PROGRAM prgBattery
VAR PERSISTENT
	bEnableBattery				: BOOL;							//{#lynus.ag#()}
	byPrioBattery				: BYTE;							//{#lynus.ag#()}
	lrMaxCapacityBattery		: LREAL;						//{#lynus.ag#()}
	lrCounterBattProd			: LREAL;						//{#lynus.ag#()}
	lrCounterBattCons			: LREAL;						//{#lynus.ag#()}
	str_IP						: STRING(15):='10.11.90.140';
	m_manual_LoadLimiting: BOOL :=TRUE;
	real_Max_ChargePower: REAL := 30000;
END_VAR
VAR
	fbBattery					: FB_Xelectrix_Powerbox_v2T;
	fbBattCounter				: FB_EnergyCounter;
	bIsEnabledBattery			: BOOL;							//{#lynus.ag#()}
	bResetBattery				: BOOL;							//{#lynus.ag#()}
	bSResetBattery				: BOOL;							//{#lynus.ag#()}
	byErrorWarningBattery		: BYTE;							//{#lynus.ag#()}
	dwSOCBattery				: DWORD;						//{#lynus.ag#()}
	rTargetPowerBattery			: REAL;							//{#lynus.ag#()}
	lrPowerBattery				: LREAL;						//{#lynus.ag#()}
	lrActualCapacityBattery		: LREAL;						//{#lynus.ag#()}
	mtest: BOOL;
	x: REAL;
	byBatteryModbusError: BOOL;									//{#lynus.ag#()}
	lrBatteryCons				: LREAL;							//{#lynus.ag#()}
	lrBatteryProd				: LREAL;							//{#lynus.ag#()}
	FB_Linear_MaxChargePower	: FB_LinearEquation;
	FB_Ramp_Max_Charging_Power	: FB_RAMP;
	FB_Linear_MaxChargePowerSOC	: FB_LinearEquation;
	
END_VAR

IF mtest THEN
	Lynus_Standards.GVL_Energy.stDataOfBatteryInverters[1,1].rTargetPowerEMS:=x;
END_IF

fbBattery(
	bEnable:= bEnableBattery, 
	bActivateControl:=TRUE , 
	byUnitID:= 1, 
	byPriority:= byPrioBattery, 
	diNrOfEMS_IN:= prgEMS.fbEMS.diNrOfEMS_OUT, 
	lrMaxCapacityBattery:= lrMaxCapacityBattery, 
	sIPAdress:= str_IP, 						// modify IP Adress
	bReset:= bResetBattery, 
	m_ManualSetpointEnable:= , 
	i_SetpointPower_Manual_kW:= , 
	m_ManualChargeDischargeMax:= m_manual_LoadLimiting, 
	r_MaxChargePower_W:= real_Max_ChargePower, 
	r_MaxDischargePower_W:= 80000, 
	stDataXelectrix=> , 
	stDataBatt=> , 
	stDataBattInverter=> , 
	stDataEMPower_Grid=> , 
	stDataEMCounter_Grid=> , 
	diNrOfBatt_OUT=> , 
	diNrOfBattInverter_OUT=> , 
	diNrOfEM_OUT_Grid=> , 
	lrMaxCapacityBattery_OUT=> , 
	iSetpointPower_Info=> );

//Out
bIsEnabledBattery := fbBattery.stDataBatt.bEnabled;
bSResetBattery := fbBattery.stDataBattInverter.bStateReset;
dwSOCBattery := fbBattery.stDataBatt.dwSOC;
rTargetPowerBattery := fbBattery.stDataBattInverter.rTargetPower;
lrPowerBattery := fbBattery.stDataBatt.lrPower;
lrActualCapacityBattery := fbBattery.lrMaxCapacityBattery_OUT;	
byErrorWarningBattery := fbBattery.stDataBatt.byErrorWarning;
byBatteryModbusError := fbBattery.stDataXelectrix.eErrorState = 1;
lrBatteryCons := fbBattery.stDataBatt.lrPowerConsumption;
lrBatteryProd := fbBattery.stDataBatt.lrPowerProduction;				
						
// EnergyCounter
fbBattCounter(
	byActiveTariff:= 1, 
	lrPowerInput:= lrPowerBattery, 
	lrTotalCounterEnergy_Consumption=> , 
	lrTotalCounterEnergy_Production=> , 
	lrCounterEnergyT1_Consumption=> , 
	lrCounterEnergyT2_Consumption=> , 
	lrCounterEnergyT1_Production=> , 
	lrCounterEnergyT2_Production=> );
	
IF fbBattCounter.lrTotalCounterEnergy_Production > lrCounterBattProd THEN  	
	lrCounterBattProd := fbBattCounter.lrTotalCounterEnergy_Production;
END_IF

IF fbBattCounter.lrTotalCounterEnergy_Consumption > lrCounterBattCons THEN  	
	lrCounterBattCons := fbBattCounter.lrTotalCounterEnergy_Consumption;
END_IF


FB_Linear_MaxChargePower(
	x1:= -40, 
	y1:= 30000, 
	x2:= -70, 
	y2:= 80000, 
	x:= LREAL_TO_REAL(prgGrid.lrPowerGrid), 
	y=>  );
FB_Linear_MaxChargePowerSOC(
	x1:= 80, 
	y1:= 80000, 
	x2:= 90, 
	y2:= 15000, 
	x:= DWORD_TO_REAL(dwSOCBattery), 
	y=>  );

FB_Ramp_Max_Charging_Power(
	realRampInput:= LIMIT(15000,FB_Linear_MaxChargePower.y,LIMIT(15000,FB_Linear_MaxChargePowerSOC.y,80000)),
	mEnableRamp:= TRUE, 
	mZeroOutput:= FALSE, 
	realRampSpeed:= 100, 
	realRampSampleTime:= 0.02 , 
	realEqualize:= 0.1, 
	realRampOutput=> real_Max_ChargePower , 
	mRampSaturised=> );

real_Max_ChargePower := LIMIT(15000,real_Max_ChargePower,80000);

END_PROGRAM

(* stored: Version 1.1.0.1, ProductVersion 3.1.4024.12
   POU prgBattery: Id {a742e2b4-8e0c-4f86-960b-eaa67f503c17}, SpecialFunc None *)
